(* PLC project Generated.project, CODESYS CODESYS V3.5 SP19 Patch 1 *)
(* stored: creationDateTime 2026-09-06T13:00:42.433406, modificationDateTime 2026-09-06T13:00:42.433406 *)

(* values of E_WinchFinalInterlockReason: NONE: Aucun blocage actif; BRAKE_COMMAND_NOT_CONFIRMED: Absence confirmation ouverture frein > 500ms; RESTART_INHIBITED: Inhibition redemarrage actif; SENSE_DROP_TIMEOUT: T_max §3bis depasse sans confirmation retombee (AC7) *)

{attribute 'qualified_only'}
{attribute 'strict'}
TYPE E_WinchFinalInterlockReason : (NONE := 0, BRAKE_COMMAND_NOT_CONFIRMED := 1, RESTART_INHIBITED := 2, SENSE_DROP_TIMEOUT := 3);
END_TYPE
